TEXTLIST TextList_xyzState
  0 = 'off'
  1 = 'idle'
  2 = 'homing'
  3 = 'ready'
  4 = 'moving'
  5 = 'stopping'
  6 = 'disabled'
  7 = 'homeTimeOut'
  100 = 'error'
   = ''
END_TEXTLIST

(* stored: Version 1.1.0.1, ProductVersion 3.1.4024.11
   TextList TextList_xyzState: Id {40e4763e-dd76-49ce-aa09-139373e3a7d0} *)
